// TIA Portal V21 export
TYPE "Std_SegnaliMacchina"
   STRUCT
      SR { S7_SetPoint := 'True'} : Array[0..1] of "Std_SendReceive";   // Send e receive
      Prm : Struct
         Watchdog : Struct   // Gestione del watchdog
            Bit : Struct   // Watchdog a bit
               Abilitato : Bool;
               RestituisciWatchdog : Bool;
               RestituisciNegato : Bool;
            END_STRUCT;
            Incrementale : Struct
               Abilitato : Bool;
            END_STRUCT;
         END_STRUCT;
         TipoComunicazione : Int;   // 0=Digitali / 1=GetPut / 2=OpcUa
      END_STRUCT;
      Allarmi : Struct
         "A" : Array[0.."K_NumAllarmiPerSegnaliMacchina"] of "Std_PrmAllarmeStd";
         WordHmi : Word;
      END_STRUCT;
   END_STRUCT;
   // // SR[0] : Send
   // // SR[1] : Receive
   // Allarmi."A"[0..3].Abilitato := FALSE;
   // Allarmi."A"[0..3].Stato := FALSE;
   // Allarmi."A"[0..3].Silenziato := FALSE;
   // Allarmi."A"[0].EnWarnHmi := FALSE;
   // Allarmi."A"[1..3].EnWarnHmi := TRUE;
   // Allarmi."A"[0..3].EnCadutaCiclo := FALSE;
END_TYPE
